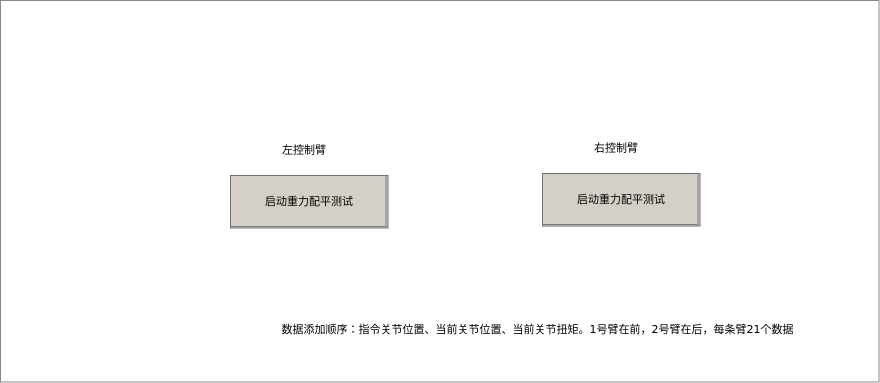
VISUALIZATION gravityTest  // 880x383
    Button (230,175 158x53), "启动重力配平测试", colour toggle: g_otherTest.g_duringMotion[1]
        tap g_otherTest.g_gravityBalanceTest[1]
    Label (229,135 150x30), "左控制臂"
    Button (542,173 158x53), "启动重力配平测试", colour toggle: g_otherTest.g_duringMotion[2]
        tap g_otherTest.g_gravityBalanceTest[2]
    Label (541,133 150x30), "右控制臂"
    Label (195,276 685x107), "数据添加顺序：指令关节位置、当前关节位置、当前关节扭矩。1号臂在前，2号臂在后，每条臂21个数据"
END_VISUALIZATION

(* stored: Version 1.1.0.1, ProductVersion 3.1.4024.11
   Visu gravityTest: Id {eff22e6a-77c2-402f-b53d-75513593854f} *)
